FUNCTION_BLOCK XtsHardware
VAR_INPUT
	Tracks : UDINT;
	TmsSwitch : ITF_TmsSwitch;
END_VAR
VAR_OUTPUT
	XtsHardwareOK : BOOL;
	Xts48VStanding : BOOL;
	Xts24VStanding : BOOL;
END_VAR
VAR
	XtsIoEnvironment : Tc3_XTS_Utility.FB_TcIoXtsEnvironment;
	bInit: BOOL;
	bMoverIdDetectionError		: BOOL;
	bMoverIdDetectionActive		: BOOL;
	bMoverIdDetected : BOOL;
	f24V: ARRAY[1..SystemParameters.nModuleNumber] OF UINT;
	f48V: ARRAY[1..SystemParameters.nModuleNumber] OF UINT;
	CurrentLive : ARRAY[1..SystemParameters.nModuleNumber] OF DINT;
	MaxCurrent : ARRAY [1..SystemParameters.nModuleNumber] OF DINT;
	nModuleCounter : UINT := 1;
	i: UDINT;
	State : XtsHardwareState;
	Logger : TcMessage_Ext;
	DetectedParts: UDINT;
	DetectedTracks : UDINT;
	DetectedModules : ARRAY[1..10] OF UDINT;
	PartIndex: UINT := 1;
	ModuleIndex : INT := 1;
	XtsHWInfo : XtsHardwareInfo;
END_VAR

IF NOT bInit THEN
	IF XtsIoEnvironment.Init(TRUE) THEN
		XtsIoEnvironment.Init(FALSE);
		bInit := TRUE;
	END_IF
	RETURN;
END_IF

CASE State OF
	XtsHardwareState.Init:
		IF GetTrackAssembly() THEN
			State := XtsHardwareState.SetDetection;
		END_IF
	
	XtsHardwareState.SetDetection:
		IF SetTracksForDetection() THEN
			State := XtsHardwareState.Redetect;
		END_IF
		
	XtsHardwareState.Redetect:
		IF TriggerMoverDetection() THEN
			State := XtsHardwareState.MoversValid;
		END_IF
		
	XtsHardwareState.MoversValid:
		IF getAllMoversValid() THEN
			State := XtsHardwareState.AllMoversFound;
		END_IF
	
	XtsHardwareState.AllMoversFound:
		IF getMoversDetected() THEN
			State := XtsHardwareState.MoverIdDetection;
		END_IF
		
	XtsHardwareState.MoverIdDetection:
		IF TriggerMoverID() THEN
			State := XtsHardwareState.XtsMode;
		END_IF
	
	XtsHardwareState.XtsMode:
		IF IsInSim() THEN
			State := XtsHardwareState.HWReady;
		ELSE
			State := XtsHardwareState.CheckModuleVoltages;
		END_IF
		
	XtsHardwareState.CheckModuleVoltages:
		Xts48VStanding := TRUE;
		Xts24VStanding := TRUE;
		FOR i := 1 TO SystemParameters.nModuleNumber DO
			IF f48V[i] < 46000 THEN
				Xts48VStanding := FALSE;
			END_IF
			IF f24V[i] < 22000 THEN
				Xts24VStanding := FALSE;
			END_IF
		END_FOR
		IF Xts24VStanding AND Xts48VStanding THEN
			State := XtsHardwareState.HWReady;
		END_IF
	
	XtsHardwareState.HWReady:
		XtsHardwareOK := TRUE;
END_CASE

getModuleInfoData();

//CYCLIC update of info
XtsHWInfo.HWState := State;

METHOD getAllMoversValid : BOOL
VAR_INPUT
END_VAR
 IF XtsIoEnvironment.XpuTcIo(1).GetAreAllPositionsValid() THEN
	 getAllMoversValid := TRUE;
	 Logger.Send(TC_EVENTS.XtsHardwareEvents.AllMoversValid,'');
 END_IF
END_METHOD

METHOD getModuleInfoData : BOOL
VAR_INPUT
END_VAR
IF XtsIoEnvironment.XpuTcIo(1).PartTcIo(PartIndex).ModuleCoE(nModuleCounter).InfoData.Update() THEN
	CurrentLive[ModuleIndex]:=XtsIoEnvironment.XpuTcIo(1).PartTcIo(PartIndex).ModuleCoE(nModuleCounter).InfoData.OverallCurrent;
	MaxCurrent[ModuleIndex]:=XtsIoEnvironment.XpuTcIo(1).PartTcIo(PartIndex).ModuleCoE(nModuleCounter).InfoData.MaxOverallCurrentLast500ms;
	f24V[ModuleIndex]:=XtsIoEnvironment.XpuTcIo(1).PartTcIo(PartIndex).ModuleCoE(nModuleCounter).InfoData.AuxiliaryVoltage24V;
	f48V[ModuleIndex]:=XtsIoEnvironment.XpuTcIo(1).PartTcIo(PartIndex).ModuleCoE(nModuleCounter).InfoData.DcLinkVoltage;
	ModuleIndex := ModuleIndex + 1;
	IF nModuleCounter = DetectedModules[PartIndex] THEN
		nModuleCounter := 1;
		IF PartIndex = DetectedParts THEN
			PartIndex := 1;
			ModuleIndex := 1;
		ELSE
			PartIndex := PartIndex + 1;
		END_IF
	ELSE
		nModuleCounter := nModuleCounter + 1;
	END_IF
END_IF
END_METHOD

METHOD PUBLIC GetMoverEnvInterface : I_TcIoXtsXpuMover
VAR_INPUT
	MoverNumber : UINT;
END_VAR
GetMoverEnvInterface := XtsIoEnvironment.XpuTcIo(1).MoverTcIo(MoverNumber);
END_METHOD

METHOD getMoversDetected : BOOL
VAR_INPUT
END_VAR
IF XtsIoEnvironment.XpuTcIo(1).GetDetectedMoverCount() = XtsIoEnvironment.XpuTcIo(1).GetExpectedMoverCount() THEN
	getMoversDetected := TRUE;
	Logger.Send(TC_EVENTS.XtsHardwareEvents.ExpectedMoversDetected,UDINT_TO_STRING(XtsIoEnvironment.XpuTcIo(1).GetExpectedMoverCount()));
ELSE
	getMoversDetected := FALSE;
	Logger.Send(TC_EVENTS.XtsHardwareEvents.ExpectedMoversNotFound,'');
END_IF
END_METHOD

METHOD PUBLIC GetTrackAssembly : BOOL
VAR_INPUT
END_VAR
DetectedTracks :=  XtsIoEnvironment.XpuTcIo(1).GetTrackCount();
IF DetectedTracks <> Tracks THEN
	Logger.Send(TC_EVENTS.XtsHardwareEvents.XtsTracksCountError,'');
	RETURN; 
END_IF
DetectedParts := XtsIoEnvironment.XpuTcIo(1).GetPartCount();
FOR i := 1 TO UDINT_TO_UINT(DetectedParts) DO
	DetectedModules[i] := XtsIoEnvironment.XpuTcIo(1).PartTcIo(1).GetModuleCount();
END_FOR
GetTrackAssembly := TRUE;

XtsHWInfo.NoOfModules := DetectedModules;
XtsHWInfo.NoOfParts := DetectedParts;
XtsHWInfo.NoOfTracks := DetectedTracks;
END_METHOD

METHOD IsInSim : BOOL
VAR_INPUT
END_VAR
IF  XtsIoEnvironment.XpuTcIo(1).GetOperationMode() = OperationMode.Simulation THEN
	IsInSim := TRUE;
	Logger.Send(TC_EVENTS.XtsHardwareEvents.XtsInSimulationMode,'');
ELSE
	IsInSim := FALSE;
END_IF
END_METHOD

METHOD SetTracksForDetection : BOOL
VAR_INPUT
END_VAR
FOR i:=1 TO XtsIoEnvironment.XpuTcIo(1).GetTrackCount() DO
	XtsIoEnvironment.XpuTcIo(1).TrackTcIo(UDINT_TO_UINT(i)).SetIsIncludedInDetection(FALSE);
END_FOR

IF XtsIoEnvironment.XpuTcIo(1).GetTrackCount() = 1 THEN
	XtsIoEnvironment.XpuTcIo(1).TrackTcIo(1).SetIsIncludedInDetection(TRUE);
	Logger.Send(TC_EVENTS.XtsHardwareEvents.ActiveTracksAddedForDetection, UDINT_TO_STRING(XtsIoEnvironment.XpuTcIo(1).GetTrackCount()));
	SetTracksForDetection := TRUE;
ELSE
	CASE TmsSwitch.Switch OF
		TmsSwitchPosition.Up: 
			XtsIoEnvironment.XpuTcIo(1).TrackTcIo(3).SetIsIncludedInDetection(TRUE);
		TmsSwitchPosition.Middle:
			XtsIoEnvironment.XpuTcIo(1).TrackTcIo(1).SetIsIncludedInDetection(TRUE);
			XtsIoEnvironment.XpuTcIo(1).TrackTcIo(2).SetIsIncludedInDetection(TRUE);
		TmsSwitchPosition.Down:
			;
	END_CASE
	Logger.Send(TC_EVENTS.XtsHardwareEvents.ActiveTracksAddedForDetection, UDINT_TO_STRING(XtsIoEnvironment.XpuTcIo(1).GetTrackCount()));
	SetTracksForDetection := TRUE;
END_IF
END_METHOD

METHOD TriggerMoverDetection : BOOL
VAR_INPUT
END_VAR
XtsIoEnvironment.XpuTcIo(1).TriggerRedetection();
Logger.Send(TC_EVENTS.XtsHardwareEvents.MoverDetectionInitiated,'');
TriggerMoverDetection := true;
END_METHOD

METHOD TriggerMoverID : BOOL
VAR_INPUT
END_VAR
// Mover1 Functionality		
// Check if "MoverIdDetectionMode" has been activated under the XtsProcessingUnit object.
IF XtsIoEnvironment.XpuTcIo(1).GetMoverIdDetectionMode() = E_MoverIdDetectionMode.Mover1
	OR XtsIoEnvironment.XpuTcIo(1).GetMoverIdDetectionMode() = 2 THEN

	// Check if the "MoverIdDetection" has already been started or the Mover1 was found.
	IF NOT (bMoverIdDetectionActive OR bMoverIdDetected) THEN
		// Trigger the "MoverIdDetection".
		XtsIoEnvironment.XpuTcIo(1).TriggerMoverIdDetection();
		Logger.Send(TC_EVENTS.XtsHardwareEvents.Mover1DetectionStarted,'');
	END_IF

	// Check for error or success of "MoverIdDetection".
	bMoverIdDetectionError 	:= XtsIoEnvironment.XpuTcIo(1).GetHasMoverIdDetectionError();
	bMoverIdDetected 	:= XtsIoEnvironment.XpuTcIo(1).GetIsMoverIdDetectionValid();
	bMoverIdDetectionActive	:= XtsIoEnvironment.XpuTcIo(1).GetIsMoverIdDetectionActive();
	
	// If the detection has an error, check for errors in output and try again.
	IF bMoverIdDetectionError THEN
		Logger.Send(TC_EVENTS.XtsHardwareEvents.Mover1DetectionFailed,'');
		RETURN; 
	END_IF

	// Do not process any further until the "MoverId" was deteced.
	IF NOT bMoverIdDetected THEN
		RETURN;
	END_IF	
	TriggerMoverID := TRUE;	
	Logger.Send(TC_EVENTS.XtsHardwareEvents.Mover1DetectionComplete,'');
ELSE
	TriggerMoverID := TRUE;
	Logger.Send(TC_EVENTS.XtsHardwareEvents.StandardMoverNumberingComplete,'');
END_IF
END_METHOD

END_FUNCTION_BLOCK

(* stored: Version 1.1.0.1, ProductVersion 3.1.4024.11
   POU XtsHardware: Id {d04838d8-bc5b-437f-a587-8af72b2fc644}, SpecialFunc None
   Method getAllMoversValid: Id {9dcfa32f-5a01-4e44-a98d-5148d4af1d1c}
   Method getModuleInfoData: Id {b00af8fa-afc5-4832-90b7-0b785a21c099}
   Method GetMoverEnvInterface: Id {41d843cc-1e86-40a6-a335-47af7a169644}
   Method getMoversDetected: Id {f316fb3e-2c49-4310-aa99-6f4cd73010f0}
   Method GetTrackAssembly: Id {86f5a3e9-8b84-41a1-b836-5c029b738ae6}
   Method IsInSim: Id {7079e35e-0b08-4e1a-90dd-d5ff9bd0268d}
   Method SetTracksForDetection: Id {51fb8179-4891-4124-a519-72890ea8063e}
   Method TriggerMoverDetection: Id {f0df76d0-8fd9-47e2-a4ee-b3636cb67c04}
   Method TriggerMoverID: Id {f94a4161-104a-471e-b20d-98cf1403fdab} *)
